Staubli VAL3: Recorder.pjx

--- Recorder.pjx ---
Parameters version=s7.6.4 stackSize=5000 millimeterUnit=true
Program file=CloseFile.pgx
Program file=OpenFile.pgx
Program file=Record.pgx
Program file=Record1.pgx
Program file=start.pgx
Program file=stop.pgx
Program file=WriteFile.pgx
Data file=Recorder.dtx

--- Recorder.dtx ---
mdesc mNomSpeed
num nFileHandle
string sFile
public bool bRecord

--- CloseFile.pgx ---
public program CloseFile()
begin
  $fileClose(nFileHandle)
  $fileClose(0)
  $fileClose(1)
  $fileClose(2)
  $fileClose(3)
  $fileClose(4)
  $fileClose(5)
  $fileClose(6)
  $fileClose(7)
  $fileClose(8)
  $fileClose(9)
end

--- Record.pgx ---
public program Record(tool x_tTool)
  local string l_sString
  local num l_ni
  local num l_nVel
  local point l_pPoint
begin
  //
  wait(bRecord==true and !isEmpty())
  l_ni=1
  l_sString=""
  do
    l_nVel=getSpeed(x_tTool)
    l_pPoint=here(x_tTool,world)
    l_sString=toString("",l_ni)+" "+toString(".1",l_nVel)+" "+toString(".2", l_pPoint.trsf.x)+" "+toString(".2", l_pPoint.trsf.y)
    l_sString=l_sString+" "+toString(".2", l_pPoint.trsf.z)
    call WriteFile(l_sString)
    l_ni=l_ni+1
    delay(0)
  until isEmpty()==true
end

--- Record1.pgx ---
public program Record1(tool x_tTool, pointRx x_pPoint, num x_nDia)
  local string l_sString
  local num l_ni
  local num l_nVel
  local point l_pPoint[3]
  local num l_nNum[3]
begin
  //
  wait(bRecord==true and !isEmpty())
  l_ni=1
  l_sString=""
  do
    l_pPoint[0]=here(x_tTool,world)
    //cmd 与半径差值
    l_nNum[0]=distance(l_pPoint[0],x_pPoint)-x_nDia/2
    //fbk与半径差值
    l_pPoint[1]=$getPosFbk(x_tTool,world)
    l_nNum[1]=distance(l_pPoint[1],x_pPoint)-x_nDia/2
    //cmd 与 fbk
    l_nNum[2]=distance(l_pPoint[0],l_pPoint[1])
    l_sString=toString(".5",l_nNum[0])+","+toString(".5",l_nNum[1])+","+toString(".5",l_nNum[2])
    call WriteFile(l_sString)
    delay(0)
  until isEmpty()==true
  bRecord=false
end

--- WriteFile.pgx ---
program WriteFile(string x_sContent)
begin
  //
  $fileSet(nFileHandle,x_sContent,1)
end
